FUNCTION_BLOCK FB_WS_Konvertierung_OLD
VAR_INPUT
	KL_Wetterstation		: KL6301;
END_VAR
VAR_OUTPUT
	Windgeschwindigkeit_Value	: REAL;
	Aussentemperatur_Value		: REAL;
	Daemmerung_Value			: REAL;
	Regensensor_Value			: REAL;
END_VAR
VAR
	Group_0_0_1			: EIB_GROUP_ADDR := (MAIN:=0,SUB_MAIN:=0,NUMBER:=1);
	Group_0_0_2			: EIB_GROUP_ADDR := (MAIN:=0,SUB_MAIN:=0,NUMBER:=2);
	Group_0_0_3			: EIB_GROUP_ADDR := (MAIN:=0,SUB_MAIN:=0,NUMBER:=3);
	Group_0_0_4			: EIB_GROUP_ADDR := (MAIN:=0,SUB_MAIN:=0,NUMBER:=4);

	Windgeschwindigkeit	: EIB_2OCTET_FLOAT_REC;
	Temperatur			: EIB_2OCTET_FLOAT_REC;
	Daemmerung			: EIB_2OCTET_FLOAT_REC;
	Regen				: EIB_2OCTET_FLOAT_REC;
END_VAR

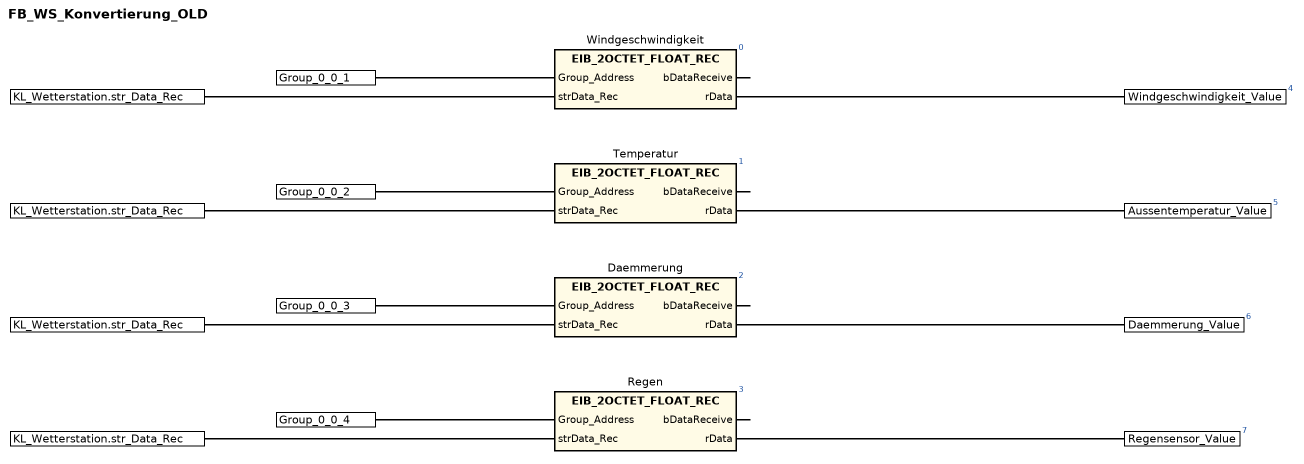
Windgeschwindigkeit(Group_Address := Group_0_0_1, strData_Rec := KL_Wetterstation.str_Data_Rec); // EIB_2OCTET_FLOAT_REC
Temperatur(Group_Address := Group_0_0_2, strData_Rec := KL_Wetterstation.str_Data_Rec); // EIB_2OCTET_FLOAT_REC
Daemmerung(Group_Address := Group_0_0_3, strData_Rec := KL_Wetterstation.str_Data_Rec); // EIB_2OCTET_FLOAT_REC
Regen(Group_Address := Group_0_0_4, strData_Rec := KL_Wetterstation.str_Data_Rec); // EIB_2OCTET_FLOAT_REC
Windgeschwindigkeit_Value := Windgeschwindigkeit.rData;
Aussentemperatur_Value := Temperatur.rData;
Daemmerung_Value := Daemmerung.rData;
Regensensor_Value := Regen.rData;

END_FUNCTION_BLOCK

(* stored: Version 1.1.0.1, ProductVersion 3.1.4024.9
   POU FB_WS_Konvertierung_OLD: Id {9e11c066-1a53-464d-8f37-2908edb17de6}, SpecialFunc None *)
